# EPICS substitutions: evrSupport/Db/ioc/IOC-LI21-BP01trig.substitutions
# Trigger records
#
# refer to Sharepoint document: Controls | Timing | timingTriggers.xls
#
# Must also have pattern records
# Note: WID, DES, TEC are in terms of nSec and are unique per device
#
file evrDevTrig.db {
#      Device	      , Description   , EVR  ,  width ,desired  , EC delay   , EVR  , EVR,  IOC          , slope
#			                            Trigger       wrt TREF   wrt fiducial loca   unit                 1/119Mhz
  pattern { DEV       ,  DESC         ,PREC  ,  WID   , DES     , TEC        , LOCA , UNIT, IOC          , ESLO
                      ,  POL          , EGU  ,  DRVL  , DRVH    , EVG        , TCTL , TPOL, TWID, TDES, CTL}
	 { BPMS:LI21:131: ,  "BPMA11"     , 0    ,  100   , 10      , LCLSBEAM   , LI21 , BP01, IOC:LI21:BP01, 8.40336692324359
                      ,  0            ,"nSec", -2.8E06, 2.8E06  IN20:EV01    , OTP0 , OT0P, OT0W, OT0D, 1 }
	 { BPMS:LI21:161: ,  "BPMA12"     , 0    ,  100   , 10      , LCLSBEAM   , LI21 , BP01, IOC:LI21:BP01, 8.40336692324359
                      ,  0            ,"nSec", -2.8E06, 2.8E06  IN20:EV01    , OTP1 , OT1P, OT1W, OT1D, 1 }
	 { BPMS:LI21:201: ,  "BPM1201"    , 0    ,  100   , 10      , LCLSBEAM   , LI21 , BP01, IOC:LI21:BP01, 8.40336692324359
                      ,  0            ,"nSec", -2.8E06, 2.8E06  IN20:EV01    , OTP2 , OT2P, OT2W, OT2D, 1 }
	 { BPMS:LI21:233: ,  "BPMS11"     , 0    ,  100   , 10      , LCLSBEAM   , LI21 , BP01, IOC:LI21:BP01, 8.40336692324359
                      ,  0            ,"nSec", -2.8E06, 2.8E06  IN20:EV01    , OTP3 , OT3P, OT3W, OT3D, 1 }
	 { BPMS:LI21:278: ,  "BPMM12"     , 0    ,  100   , 10      , LCLSBEAM   , LI21 , BP01, IOC:LI21:BP01, 8.40336692324359
                      ,  0            ,"nSec", -2.8E06, 2.8E06  IN20:EV01    , OTP4 , OT4P, OT4W, OT4D, 1 }
	 { BPMS:LI21:301: ,  "BPM1301"    , 0    ,  100   , 10      , LCLSBEAM   , LI21 , BP01, IOC:LI21:BP01, 8.40336692324359
                      ,  0            ,"nSec", -2.8E06, 2.8E06  IN20:EV01    , OTP5 , OT5P, OT5W, OT5D, 1 }
	 { BPMS:LI21:315: ,  "BPMM14"     , 0    ,  100   , 10      , LCLSBEAM   , LI21 , BP01, IOC:LI21:BP01, 8.40336692324359
                      ,  0            ,"nSec", -2.8E06, 2.8E06  IN20:EV01    , OTP6 , OT6P, OT6W, OT6D, 1 }
{ BPMS:LI21:131:CALB  ,  "BPMA11 Calb", 0    ,  100   , 10      , TS5_120_   , LI21 , BP01, IOC:LI21:BP01, 8.40336692324359
                      ,  0            ,"nSec", -2.8E06, 2.8E06  IN20:EV01    , OTP7 , OT7P, OT7W, OT7D, 1 }
{ BPMS:LI21:161:CALB  ,  "BPMA12 Calb", 0    ,  100   , 10      , TS5_120_   , LI21 , BP01, IOC:LI21:BP01, 8.40336692324359
                      ,  0            ,"nSec", -2.8E06, 2.8E06  IN20:EV01    , OTP8 , OT8P, OT8W, OT8D, 1 }
{ BPMS:LI21:201:CALB  ,  "BPM1201 Calb",0    ,  100   , 10      , TS5_120_   , LI21 , BP01, IOC:LI21:BP01, 8.40336692324359
                      ,  0            ,"nSec", -2.8E06, 2.8E06  IN20:EV01    , OTP9 , OT9P, OT9W, OT9D, 1 }
{ BPMS:LI21:233:CALB  ,  "BPMS11 Calb", 0    ,  100   , 10      , TS5_120_   , LI21 , BP01, IOC:LI21:BP01, 8.40336692324359
                      ,  0            ,"nSec", -2.8E06, 2.8E06  IN20:EV01    , OTPA , OTAP, OTAW, OTAD, 1 }
{ BPMS:LI21:278:CALB  ,  "BPMM12 Calb", 0    ,  100   , 10      , TS5_120_   , LI21 , BP01, IOC:LI21:BP01, 8.40336692324359
                      ,  0            ,"nSec", -2.8E06, 2.8E06  IN20:EV01    , OTPB , OTBP, OTBW, OTBD, 1 }
{ BPMS:LI21:301:CALB  ,  "BPM1301 Calb",0    ,  100   , 10      , TS5_120_   , LI21 , BP01, IOC:LI21:BP01, 8.40336692324359
                      ,  0            ,"nSec", -2.8E06, 2.8E06  IN20:EV01    , OTPC , OTCP, OTCW, OTCD, 1 }
{ BPMS:LI21:315:CALB  ,  "BPMM14 Calb", 0    ,  100   , 10      , TS5_120_   , LI21 , BP01, IOC:LI21:BP01, 8.40336692324359
                      ,  0            ,"nSec", -2.8E06, 2.8E06  IN20:EV01    , OTPD , OTDP, OTDW, OTDD, 1 }
# spare triggers 1-5, FP (VME)
	 { TRIG:LI21:BP01:, "Spare Trig 1", 0    ,  100   , 10      , TS5_120_   , LI21 , BP01, IOC:LI21:BP01, 8.40336692324359
                      ,  0            ,"nSec", -2.8E06, 2.8E06  , LI21:EV01  , DG0E , DG0P, DG0W, DG0D, 1 }
	 { TRIG:LI21:BP02:, "Spare Trig 2", 0    ,  100   , 10      , TS5_120_   , LI21 , BP01, IOC:LI21:BP01, 8.40336692324359
                      ,  0            ,"nSec", -2.8E06, 2.8E06  , LI21:EV01  , DG1E , DG1P, DG0W, DG1D, 1 }
	 { TRIG:LI21:BP03:, "Spare Trig 3", 0    ,  100   , 10      , TS5_120_   , LI21 , BP01, IOC:LI21:BP01, 8.40336692324359
                      ,  0            ,"nSec", -2.8E06, 2.8E06  , LI21:EV01  , DG2E , DG2P, DG2W, DG2D, 1 }
	 { TRIG:LI21:BP04:, "Spare Trig 4", 0    ,  100   , 10      , TS5_120_   , LI21 , BP01, IOC:LI21:BP01, 8.40336692324359
                      ,  0            ,"nSec", -2.8E06, 2.8E06  , LI21:EV01  , DG3E , DG3P, DG3W, DG3D, 1 }
	 { TRIG:LI21:BP05:, "Spare Trig 5", 0    ,  100   , 10      , TS5_120_   , LI21 , BP01, IOC:LI21:BP01, 8.40336692324359
                      ,  0            ,"nSec", -2.8E06, 2.8E06  , LI21:EV01  , DG4E , DG4P, DG4W, DG4D, 1 }

}
